(* CoDeSys 2.3.9.28 project: md_roman_5.pro *)
(* Libraries: SysLibTime.lib 2.12.10 13:48:32, Building_common.lib 2.12.10 13:48:40, mod_com.lib 2.12.10 13:48:32, DaylightSaving.lib 2.12.10 13:48:32, PowerMeasurement_01.lib 28.1.08 13:32:32, ModbusEthernet_04.lib 2.12.10 13:48:36, Util.lib 18.5.10 14:14:28, Standard.lib 2.12.10 13:48:34, SYSLIBCALLBACK.LIB 2.12.10 13:48:32, SysLibRtc.lib 2.12.10 13:48:32, SysLibFile.lib 2.12.10 13:48:34, Visu_Scheduler_03_e.lib 15.3.11 07:49:24, Scheduler_03.lib 9.3.11 15:45:22, DALI_02.lib 19.10.11 13:30:12, WagoLibDaylightSaving.lib 2.12.10 13:48:32, Ethernet.lib 2.12.10 13:48:32 *)

(* PLC configuration (modules and I/O channels)
TL01 AT %IX17.0 [BOOLOnX_I] Vypinac_sklad_sklad
TL02 AT %IX17.1 [BOOLOnX_I] Vypinac_sklad_prodejna
TL03 AT %IX17.2 [BOOLOnX_I] Vypinac_sklad_z_venku
TL04 AT %IX17.3 [BOOLOnX_I] Vypinac_sklad_vrata_predni
TL05 AT %IX17.4 [BOOLOnX_I] Vypinac_sklad_vrata_zadni
TL06 AT %IX17.5 [BOOLOnX_I] Vypinac_prodejna_kolotoc_sude
TL07 AT %IX17.6 [BOOLOnX_I] Vypinac_prodejna_kolotoc_liche
TL08 AT %IX17.7 [BOOLOnX_I] Vypinac_prodejna_vypinac
TL09 AT %IX17.8 [BOOLOnX_I] Prodejna_Dali
TL10 AT %IX17.9 [BOOLOnX_I] Prodejna_faugule_OUT13
TL11 AT %IX17.10 [BOOLOnX_I] Ch_3 Digital input
TL12 AT %IX17.11 [BOOLOnX_I] Ch_4 Digital input
TL13 AT %IX17.12 [BOOLOnX_I] Ch_5 Digital input
AT %IX17.13 [BOOLOnX_I] Ch_6 Digital input
AT %IX17.14 [BOOLOnX_I] Ch_7 Digital input
AT %IX17.15 [BOOLOnX_I] Ch_8 Digital input
AT %IX18.0 [BOOLOnX_I] Ch_1 Digital input
AT %IX18.1 [BOOLOnX_I] Ch_2 Digital input
AT %IX18.2 [BOOLOnX_I] Ch_3 Digital input
AT %IX18.3 [BOOLOnX_I] Ch_4 Digital input
AT %IX18.4 [BOOLOnX_I] Ch_5 Digital input
AT %IX18.5 [BOOLOnX_I] Ch_6 Digital input
AT %IX18.6 [BOOLOnX_I] Ch_7 Digital input
AT %IX18.7 [BOOLOnX_I] Ch_8 Digital input
KA01 AT %QX9.0 [BOOLOnX_Q] Nevim
KA02 AT %QX9.1 [BOOLOnX_Q] kolotoc2
KA03 AT %QX9.2 [BOOLOnX_Q] kolotoc3
KA04 AT %QX9.3 [BOOLOnX_Q] kolotoc4
KA05 AT %QX9.4 [BOOLOnX_Q] kolotoc5
KA06 AT %QX9.5 [BOOLOnX_Q] kolotoc6
KA07 AT %QX9.6 [BOOLOnX_Q] kolotoc7
KA08 AT %QX9.7 [BOOLOnX_Q] kolotoc8
0750-0530 8 DO 24 V DC 0.5A [Type_10_8_Channels] node 4, in %IB4 out %QB4 {INTTypePAAssignment = PLC; INTTypeModule = plugged}
  KA09 AT %QX9.8 [BOOLOnX_Q] kolotoc9
  KA10 AT %QX9.9 [BOOLOnX_Q] kolotoc10
  KA11 AT %QX9.10 [BOOLOnX_Q] kolotoc11
  KA12 AT %QX9.11 [BOOLOnX_Q] kolotoc12
  KA13 AT %QX9.12 [BOOLOnX_Q] svetlo_vchod_do_prodejny
  KA14 AT %QX9.13 [BOOLOnX_Q] reklama
  KA15 AT %QX9.14 [BOOLOnX_Q] svetlo_vrata_predni
  KA16 AT %QX9.15 [BOOLOnX_Q] svetlo_vrata_zadni
0750-0530 8 DO 24 V DC 0.5A [Type_10_8_Channels] node 5, in %IB5 out %QB5 {INTTypePAAssignment = PLC; INTTypeModule = plugged}
  KA17 AT %QX10.0 [BOOLOnX_Q] Ch_1 Digital output
  AT %QX10.1 [BOOLOnX_Q] Ch_2 Digital output
  AT %QX10.2 [BOOLOnX_Q] Ch_3 Digital output
  KA20 AT %QX10.3 [BOOLOnX_Q] Ch_4 Digital output
  AT %QX10.4 [BOOLOnX_Q] Ch_5 Digital output
  AT %QX10.5 [BOOLOnX_Q] Ch_6 Digital output
  AT %QX10.6 [BOOLOnX_Q] Ch_7 Digital output
  AT %QX10.7 [BOOLOnX_Q] Ch_8 Digital output
0750-0530 8 DO 24 V DC 0.5A [Type_10_8_Channels] node 6, in %IB6 out %QB6 {INTTypePAAssignment = PLC; INTTypeModule = plugged}
  AT %QX10.8 [BOOLOnX_Q] Ch_1 Digital output
  AT %QX10.9 [BOOLOnX_Q] Ch_2 Digital output
  AT %QX10.10 [BOOLOnX_Q] Ch_3 Digital output
  AT %QX10.11 [BOOLOnX_Q] Ch_4 Digital output
  AT %QX10.12 [BOOLOnX_Q] Ch_5 Digital output
  AT %QX10.13 [BOOLOnX_Q] Ch_6 Digital output
  AT %QX10.14 [BOOLOnX_Q] Ch_7 Digital output
  AT %QX10.15 [BOOLOnX_Q] Ch_8 Digital output
Analog_1 AT %IW0 [WORDOnW_I] Ch_1 Input word
AT %IW1 [WORDOnW_I] Ch_2 Input word
AT %IW2 [WORDOnW_I] Ch_3 Input word
AT %IW3 [WORDOnW_I] Ch_4 Input word
0750-0460/0000-0005 4 AI NI1000 (RTD) [Type_44_4_Channels] node 8, in %IB8 out %QB8 {INTTypePAAssignment = PLC; INTTypeModule = plugged}
  Teplota_1 AT %IW4 [INTOnW_I] Ch_1 signed Input value
  Teplota_2 AT %IW5 [INTOnW_I] Ch_2 signed Input value
  Teplota_3 AT %IW6 [INTOnW_I] Ch_3 signed Input value
  Teplota_4 AT %IW7 [INTOnW_I] Ch_4 signed Input value
0750-0641 DALI/DSI-Master [Type_36_1_Channels] node 9, in %IB9 out %QB9 {INTTypePAAssignment = PLC; INTTypeModule = plugged}
  AT %IX8.0 [BOOLOnX_I] Transmit accepted
  AT %IX8.1 [BOOLOnX_I] Receive request
  AT %IX8.2 [BOOLOnX_I] Init accepted
  AT %IX8.3 [BOOLOnX_I] Actor Error
  AT %IX8.4 [BOOLOnX_I] Frame Error
  AT %IX8.5 [BOOLOnX_I] Bus Error
  AT %IX8.6 [BOOLOnX_I] General Module Error
  AT %IB17 [BYTEOnB_I] DALI Response
  AT %IB18 [BYTEOnB_I] DALI Address
  AT %IB19 [BYTEOnB_I] Message 3
  AT %IB20 [BYTEOnB_I] Message 2
  AT %IB21 [BYTEOnB_I] Message 1
  AT %QX0.0 [BOOLOnX_Q] Transmit request
  AT %QX0.1 [BOOLOnX_Q] Receive accepted
  AT %QX0.2 [BOOLOnX_Q] Init request
  AT %QB1 [BYTEOnB_Q] DALI Command, DSI dimming value
  AT %QB2 [BYTEOnB_Q] DALI Address
  AT %QB3 [BYTEOnB_Q] Parameter 2
  AT %QB4 [BYTEOnB_Q] Parameter 1
  AT %QB5 [BYTEOnB_Q] Command extension
fazeVstup AT %IB22 [BYTEOnB_I] First Byte of 12
fazeVystup AT %QB6 [BYTEOnB_Q] First Byte of 12
Fieldbus variables [FB_VARS] node 1, in %IB0 out %QB0
*)

(* Task configuration *)
TASK hlavni (PRIORITY := 1, INTERVAL := T#20ms);
	PLC_PRG();
END_TASK
TASK Cas (PRIORITY := 15, INTERVAL := T#1000ms);
	LetniZimniCas();
	CasProg();
END_TASK

(* Global variable list: Global_Variables *)
VAR_GLOBAL
	start_bit: BOOL;
	Inicialiazace_DALI: BOOL;
	Inicializuj: BOOL;
	TL08s: BOOL;
	TL07s: BOOL;
	TL10s: BOOL;
	TL06s: BOOL;
	TL05s: BOOL;
	TL01s: BOOL;
	TL09s: BOOL;
	Cidlo: REAL;
	Uroven1: REAL := 3.5;
	Uroven2: REAL := 5;
	ZpozdeniCidla: BYTE := 10;
	Cidlo_zpozdene: REAL;

	CasDatumAktualni 	: DT;
	DenvTydnu			: BYTE;
	Leto 					: BOOL;
	sCasDatumAktualni 	: STRING[20];

	Uroven_reklama1: REAL := 1.5;

	VzdalenyVstup1: BOOL;
	VzdalenyVstup2: BOOL;
	VzdalenyVstup3: BOOL;
	VzdalenyVstup4: BOOL;
	VzdalenyVstup5: BOOL;
	VzdalenyVstup6: BOOL;
	VzdalenyVstup7: BOOL;
	VzdalenyVstup8: BOOL;
	VzdalenyVstup9: BOOL;
	VzdalenyVstup10: BOOL;
	VzdalenyVstup11: BOOL;
	VzdalenyVstup12: BOOL;
	VzdalenyVstup13: BOOL;
	VzdalenyVstup14: BOOL;
	VzdalenyVstup15: BOOL;
	VzdalenyVstup16: BOOL;

	VzdalenyVystup1: BOOL;
	VzdalenyVystup2: BOOL;
	VzdalenyVystup3: BOOL;
	VzdalenyVystup4: BOOL;
	VzdalenyVystup5: BOOL;
	VzdalenyVystup6: BOOL;
	VzdalenyVystup7: BOOL;
	VzdalenyVystup8: BOOL;
	VzdalenyVystup9: BOOL;
	VzdalenyVystup10: BOOL;
	VzdalenyVystup11: BOOL;
	VzdalenyVystup12: BOOL;
	VzdalenyVystup13: BOOL;
	VzdalenyVystup14: BOOL;
	VzdalenyVystup15: BOOL;
	VzdalenyVystup16: BOOL;

	VzdalenaTeplota1: WORD;
	VzdalenaTeplota2: WORD;
	VzdalenaTeplota3: WORD;
	VzdalenaTeplota4: WORD;

	IPSlaveProdejnaMaterial: STRING:= '192.168.111.202';

	INVnitrniSvetla1: BOOL;
	INVnitrniSvetla2: BOOL;
	INVnitrniSvetla3: BOOL;
	INVnitrniZasuvkyDenniProvoz: BOOL;
	INSvetloNadVchodem: BOOL;
	INVnitrniReklama: BOOL;
	INVenkovniReklama: BOOL;
	INTopeniOkap: BOOL;
	OUTVnitrniSvetla1: BOOL;		(*KA1*)
	OUTVnitrniSvetla2: BOOL;		(*KA2*)
	OUTVnitrniSvetla3: BOOL;		(*KA3*)
	OUTVnitrniReklama: BOOL;		(*KA4*)
	OUTVenkovniReklama1: BOOL;		(*KA5*)
	OUTVenkovniReklama2: BOOL;		(*KA6*)
	OUTVenkovniReklama3: BOOL;		(*KA7*)
	OUTSvetloNadVchodem: BOOL;		(*KA78*)
	OUTTopeniOkap1: BOOL;		(*KA9*)
	OUTTopeniOkap2: BOOL;		(*KA10*)
	OUTZasuvky1: BOOL;		(*KA11*)
	OUTZasuvky3: BOOL;		(*KA12*)
	OUTNouzoveOsvetleni: BOOL;		(*KA13*)
	OUTVnitrniZasuvkyDenniProvoz: BOOL;
	OUTVenkovniReklama: BOOL;
	OUTTopeniOkap: BOOL;

	INVenkovniTeplota: REAL;
END_VAR
VAR_GLOBAL RETAIN PERSISTENT
	typCasProg1: typScheduleWeekly;
	typCasProg2: typScheduleWeekly;

	typCasProg3: typScheduleWeekly;
	typCasProg4: typScheduleWeekly;

	typCasProg5: typScheduleWeekly;
	typCasProg6: typScheduleWeekly;
END_VAR

(* POU PLC_PRG, FBD *)
PROGRAM PLC_PRG
VAR
	cas_datum: CurTimeEx;
	System_cas: SysTime64;
	System_datum: SystemTimeDate;
	kolotoc1: kolotoc;
	kolotoc2: kolotoc;
	BLINK_nouzaky: BLINK;
	LibovolnyVystup: BOOL;
	komunikace: SlaveUDP_IO;

	Test: SlaveUDP_IO;
	sendStr: ARRAY [1..100] OF WORD;
	RecStr: ARRAY [1..100] OF WORD;

	Init: BOOL;
	NoError: BOOL;

	VzdaleneVstupy1: WORD_TO_BOOL_16b;
	VzdaleneVystupy1: BOOL_TO_WORD_16b;
END_VAR
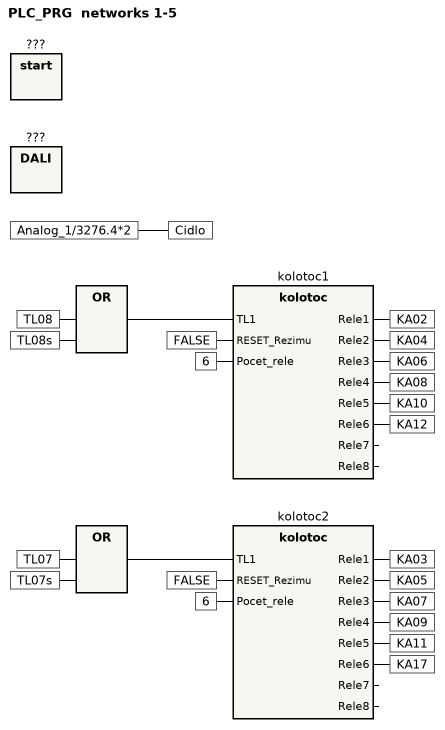
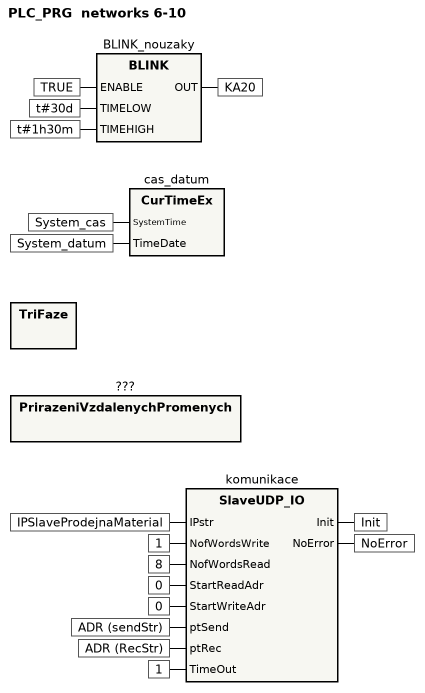
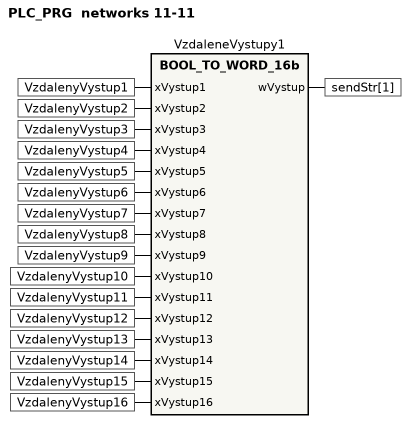
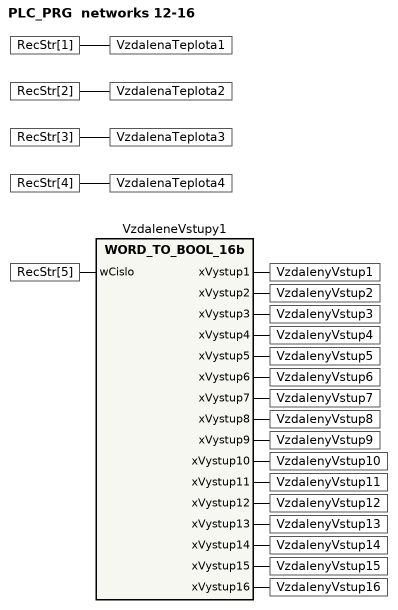
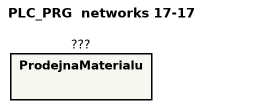
_FBD_ (* Function Block Diagram *)
NETWORK 1
	???:start()
NETWORK 2
	???:DALI()
NETWORK 3
	Analog_1/3276.4*2 => Cidlo
NETWORK 4
	kolotoc1:kolotoc(TL1: OR(TL08, TL08s), RESET_Rezimu: FALSE, Pocet_rele: 6, Rele2 => KA04, Rele3 => KA06, Rele4 => KA08, Rele5 => KA10, Rele6 => KA12) => KA02
NETWORK 5
	kolotoc2:kolotoc(TL1: OR(TL07, TL07s), RESET_Rezimu: FALSE, Pocet_rele: 6, Rele2 => KA05, Rele3 => KA07, Rele4 => KA09, Rele5 => KA11, Rele6 => KA17) => KA03
NETWORK 6
	BLINK_nouzaky:BLINK(ENABLE: TRUE, TIMELOW: t#30d, TIMEHIGH: t#1h30m) => KA20
NETWORK 7
	cas_datum:CurTimeEx(SystemTime: System_cas, TimeDate: System_datum)
NETWORK 8
	TriFaze()
NETWORK 9
	???:PrirazeniVzdalenychPromenych()
NETWORK 10
	komunikace:SlaveUDP_IO(IPstr: IPSlaveProdejnaMaterial, NofWordsWrite: 1, NofWordsRead: 8, StartReadAdr: 0, StartWriteAdr: 0, ptSend: ADR (sendStr), ptRec: ADR (RecStr), TimeOut: 1, NoError => NoError) => Init
NETWORK 11
	VzdaleneVystupy1:BOOL_TO_WORD_16b(xVystup1: VzdalenyVystup1, xVystup2: VzdalenyVystup2, xVystup3: VzdalenyVystup3, xVystup4: VzdalenyVystup4, xVystup5: VzdalenyVystup5, xVystup6: VzdalenyVystup6, xVystup7: VzdalenyVystup7, xVystup8: VzdalenyVystup8, xVystup9: VzdalenyVystup9, xVystup10: VzdalenyVystup10, xVystup11: VzdalenyVystup11, xVystup12: VzdalenyVystup12, xVystup13: VzdalenyVystup13, xVystup14: VzdalenyVystup14, xVystup15: VzdalenyVystup15, xVystup16: VzdalenyVystup16) => sendStr[1]
NETWORK 12
	RecStr[1] => VzdalenaTeplota1
NETWORK 13
	RecStr[2] => VzdalenaTeplota2
NETWORK 14
	RecStr[3] => VzdalenaTeplota3
NETWORK 15
	RecStr[4] => VzdalenaTeplota4
NETWORK 16
	VzdaleneVstupy1:WORD_TO_BOOL_16b(wCislo: RecStr[5], xVystup2 => VzdalenyVstup2, xVystup3 => VzdalenyVstup3, xVystup4 => VzdalenyVstup4, xVystup5 => VzdalenyVstup5, xVystup6 => VzdalenyVstup6, xVystup7 => VzdalenyVstup7, xVystup8 => VzdalenyVstup8, xVystup9 => VzdalenyVstup9, xVystup10 => VzdalenyVstup10, xVystup11 => VzdalenyVstup11, xVystup12 => VzdalenyVstup12, xVystup13 => VzdalenyVstup13, xVystup14 => VzdalenyVstup14, xVystup15 => VzdalenyVstup15, xVystup16 => VzdalenyVstup16) => VzdalenyVstup1
NETWORK 17
	???:ProdejnaMaterialu()
_END_FBD_
(* the same logic as Structured Text *)
(* Network 1: see the listing above *)
(* Network 2: see the listing above *)
(* Network 3 *)
Cidlo := Analog_1/3276.4*2;
(* Network 4 *)
kolotoc1(TL1 := TL08 OR TL08s, RESET_Rezimu := FALSE, Pocet_rele := 6);
KA04 := kolotoc1.Rele2;
KA06 := kolotoc1.Rele3;
KA08 := kolotoc1.Rele4;
KA10 := kolotoc1.Rele5;
KA12 := kolotoc1.Rele6;
KA02 := kolotoc1.Rele1;
(* Network 5 *)
kolotoc2(TL1 := TL07 OR TL07s, RESET_Rezimu := FALSE, Pocet_rele := 6);
KA05 := kolotoc2.Rele2;
KA07 := kolotoc2.Rele3;
KA09 := kolotoc2.Rele4;
KA11 := kolotoc2.Rele5;
KA17 := kolotoc2.Rele6;
KA03 := kolotoc2.Rele1;
(* Network 6 *)
BLINK_nouzaky(ENABLE := TRUE, TIMELOW := t#30d, TIMEHIGH := t#1h30m);
KA20 := BLINK_nouzaky.OUT;
(* Network 7 *)
cas_datum(SystemTime := System_cas, TimeDate := System_datum);
(* Network 8 *)
TriFaze();
(* Network 9: see the listing above *)
(* Network 10 *)
komunikace(IPstr := IPSlaveProdejnaMaterial, NofWordsWrite := 1, NofWordsRead := 8, StartReadAdr := 0, StartWriteAdr := 0, ptSend := ADR (sendStr), ptRec := ADR (RecStr), TimeOut := 1);
NoError := komunikace.NoError;
Init := komunikace.Init;
(* Network 11 *)
VzdaleneVystupy1(xVystup1 := VzdalenyVystup1, xVystup2 := VzdalenyVystup2, xVystup3 := VzdalenyVystup3, xVystup4 := VzdalenyVystup4, xVystup5 := VzdalenyVystup5, xVystup6 := VzdalenyVystup6, xVystup7 := VzdalenyVystup7, xVystup8 := VzdalenyVystup8, xVystup9 := VzdalenyVystup9, xVystup10 := VzdalenyVystup10, xVystup11 := VzdalenyVystup11, xVystup12 := VzdalenyVystup12, xVystup13 := VzdalenyVystup13, xVystup14 := VzdalenyVystup14, xVystup15 := VzdalenyVystup15, xVystup16 := VzdalenyVystup16);
sendStr[1] := VzdaleneVystupy1.wVystup;
(* Network 12 *)
VzdalenaTeplota1 := RecStr[1];
(* Network 13 *)
VzdalenaTeplota2 := RecStr[2];
(* Network 14 *)
VzdalenaTeplota3 := RecStr[3];
(* Network 15 *)
VzdalenaTeplota4 := RecStr[4];
(* Network 16 *)
VzdaleneVstupy1(wCislo := RecStr[5]);
VzdalenyVstup2 := VzdaleneVstupy1.xVystup2;
VzdalenyVstup3 := VzdaleneVstupy1.xVystup3;
VzdalenyVstup4 := VzdaleneVstupy1.xVystup4;
VzdalenyVstup5 := VzdaleneVstupy1.xVystup5;
VzdalenyVstup6 := VzdaleneVstupy1.xVystup6;
VzdalenyVstup7 := VzdaleneVstupy1.xVystup7;
VzdalenyVstup8 := VzdaleneVstupy1.xVystup8;
VzdalenyVstup9 := VzdaleneVstupy1.xVystup9;
VzdalenyVstup10 := VzdaleneVstupy1.xVystup10;
VzdalenyVstup11 := VzdaleneVstupy1.xVystup11;
VzdalenyVstup12 := VzdaleneVstupy1.xVystup12;
VzdalenyVstup13 := VzdaleneVstupy1.xVystup13;
VzdalenyVstup14 := VzdaleneVstupy1.xVystup14;
VzdalenyVstup15 := VzdaleneVstupy1.xVystup15;
VzdalenyVstup16 := VzdaleneVstupy1.xVystup16;
VzdalenyVstup1 := VzdaleneVstupy1.xVystup1;
(* Network 17: see the listing above *)
END_PROGRAM

(* POU dali/kolotoc, FBD *)
FUNCTION_BLOCK kolotoc
VAR
	Data_platna: BOOL;
	Data_platna_reset: BOOL;
	T_Data_platna: TON;
	T_Data_platna_reset: TON;
	Stisk_kratky: BOOL := FALSE;
	Stisk_dlouhy: BOOL := FALSE;
	T_stisk_TLx: TON;
	F_trig_hr1: F_TRIG;
	R_trig_hr2: R_TRIG;
	TL1_Citac: CTU;
	SR_stisk_TLx: SR;
	ZAP_VYP: BOOL;




	TP_byl_kratky: TP;
	Q_byl_kratky: BOOL;
	blok_kratky: BOOL;
	TL1_hr1: BOOL;
	SET_stisk_TL1: BOOL;
	Q_stisk_TL1: BOOL;
	TL1_INT: INT;
END_VAR

VAR_OUTPUT
	Rele1: BOOL;
	Rele2: BOOL;
	Rele3: BOOL;
	Rele4: BOOL;
	Rele5: BOOL;
	Rele6: BOOL;
	Rele7: BOOL;
	Rele8: BOOL;
END_VAR
VAR_INPUT
	TL1: BOOL;
	RESET_Rezimu: BOOL;
	Pocet_rele: INT;
END_VAR
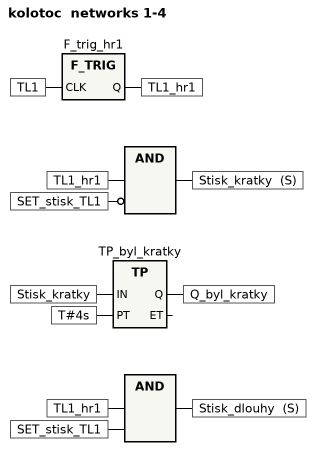
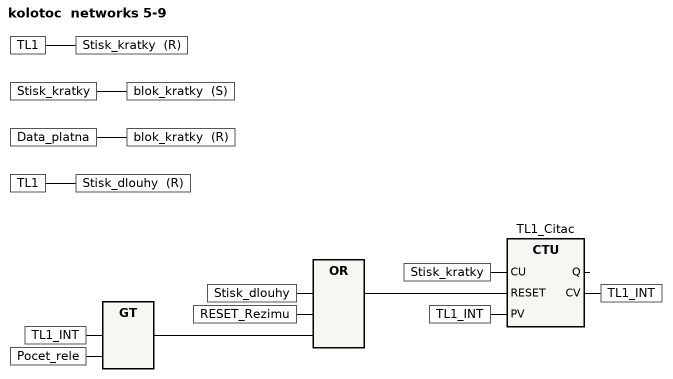
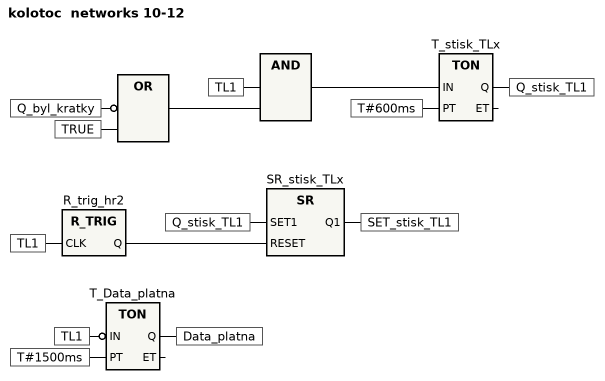
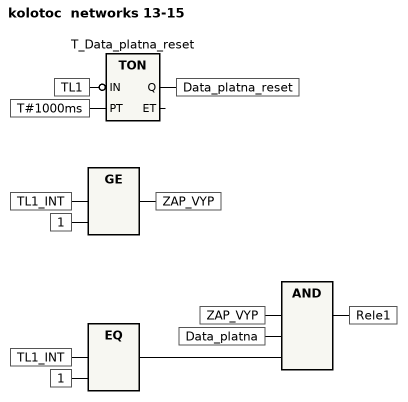
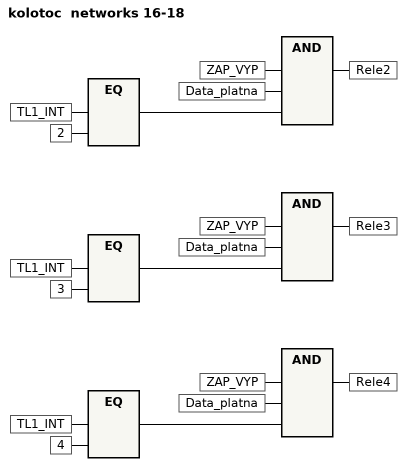
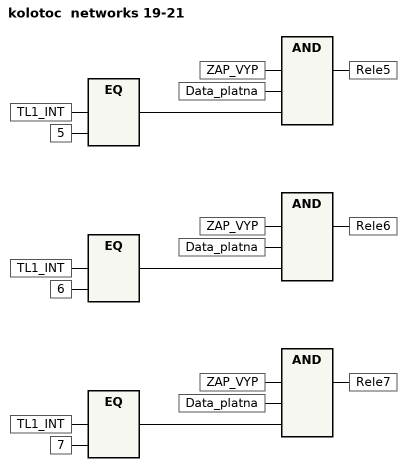
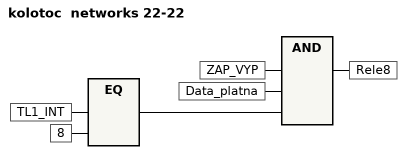
_FBD_ (* Function Block Diagram *)
NETWORK 1
	F_trig_hr1:F_TRIG(CLK: TL1) => TL1_hr1
NETWORK 2
	AND(TL1_hr1, NOT SET_stisk_TL1) => S Stisk_kratky
NETWORK 3
	TP_byl_kratky:TP(IN: Stisk_kratky, PT: T#4s) => Q_byl_kratky
NETWORK 4
	AND(TL1_hr1, SET_stisk_TL1) => S Stisk_dlouhy
NETWORK 5
	TL1 => R Stisk_kratky
NETWORK 6
	Stisk_kratky => S blok_kratky
NETWORK 7
	Data_platna => R blok_kratky
NETWORK 8
	TL1 => R Stisk_dlouhy
NETWORK 9
	TL1_Citac:CTU(CU: Stisk_kratky, RESET: OR(Stisk_dlouhy, RESET_Rezimu, GT(TL1_INT, Pocet_rele)), PV: TL1_INT, CV => TL1_INT)
NETWORK 10 (* delka stisku TLx *)
	T_stisk_TLx:TON(IN: AND(TL1, OR(NOT Q_byl_kratky, TRUE)), PT: T#600ms) => Q_stisk_TL1
NETWORK 11
	SR_stisk_TLx:SR(SET1: Q_stisk_TL1, RESET: R_trig_hr2:R_TRIG(CLK: TL1)) => SET_stisk_TL1
NETWORK 12 (* Data platna *)
	T_Data_platna:TON(IN: NOT TL1, PT: T#1500ms) => Data_platna
NETWORK 13 (* Data platna *)
	T_Data_platna_reset:TON(IN: NOT TL1, PT: T#1000ms) => Data_platna_reset
NETWORK 14
	GE(TL1_INT, 1) => ZAP_VYP
NETWORK 15
	AND(ZAP_VYP, Data_platna, EQ(TL1_INT, 1)) => Rele1
NETWORK 16
	AND(ZAP_VYP, Data_platna, EQ(TL1_INT, 2)) => Rele2
NETWORK 17
	AND(ZAP_VYP, Data_platna, EQ(TL1_INT, 3)) => Rele3
NETWORK 18
	AND(ZAP_VYP, Data_platna, EQ(TL1_INT, 4)) => Rele4
NETWORK 19
	AND(ZAP_VYP, Data_platna, EQ(TL1_INT, 5)) => Rele5
NETWORK 20
	AND(ZAP_VYP, Data_platna, EQ(TL1_INT, 6)) => Rele6
NETWORK 21
	AND(ZAP_VYP, Data_platna, EQ(TL1_INT, 7)) => Rele7
NETWORK 22
	AND(ZAP_VYP, Data_platna, EQ(TL1_INT, 8)) => Rele8
_END_FBD_
(* the same logic as Structured Text *)
(* Network 1 *)
F_trig_hr1(CLK := TL1);
TL1_hr1 := F_trig_hr1.Q;
(* Network 2 *)
IF TL1_hr1 AND NOT SET_stisk_TL1 THEN Stisk_kratky := TRUE; END_IF;
(* Network 3 *)
TP_byl_kratky(IN := Stisk_kratky, PT := T#4s);
Q_byl_kratky := TP_byl_kratky.Q;
(* Network 4 *)
IF TL1_hr1 AND SET_stisk_TL1 THEN Stisk_dlouhy := TRUE; END_IF;
(* Network 5 *)
IF TL1 THEN Stisk_kratky := FALSE; END_IF;
(* Network 6 *)
IF Stisk_kratky THEN blok_kratky := TRUE; END_IF;
(* Network 7 *)
IF Data_platna THEN blok_kratky := FALSE; END_IF;
(* Network 8 *)
IF TL1 THEN Stisk_dlouhy := FALSE; END_IF;
(* Network 9 *)
TL1_Citac(CU := Stisk_kratky, RESET := Stisk_dlouhy OR RESET_Rezimu OR (TL1_INT > Pocet_rele), PV := TL1_INT);
TL1_INT := TL1_Citac.CV;
(* Network 10: see the listing above *)
(* Network 11 *)
R_trig_hr2(CLK := TL1);
SR_stisk_TLx(SET1 := Q_stisk_TL1, RESET := R_trig_hr2.Q);
SET_stisk_TL1 := SR_stisk_TLx.Q1;
(* Network 12 *)
T_Data_platna(IN := NOT TL1, PT := T#1500ms);
Data_platna := T_Data_platna.Q;
(* Network 13 *)
T_Data_platna_reset(IN := NOT TL1, PT := T#1000ms);
Data_platna_reset := T_Data_platna_reset.Q;
(* Network 14 *)
ZAP_VYP := TL1_INT >= 1;
(* Network 15 *)
Rele1 := ZAP_VYP AND Data_platna AND (TL1_INT = 1);
(* Network 16 *)
Rele2 := ZAP_VYP AND Data_platna AND (TL1_INT = 2);
(* Network 17 *)
Rele3 := ZAP_VYP AND Data_platna AND (TL1_INT = 3);
(* Network 18 *)
Rele4 := ZAP_VYP AND Data_platna AND (TL1_INT = 4);
(* Network 19 *)
Rele5 := ZAP_VYP AND Data_platna AND (TL1_INT = 5);
(* Network 20 *)
Rele6 := ZAP_VYP AND Data_platna AND (TL1_INT = 6);
(* Network 21 *)
Rele7 := ZAP_VYP AND Data_platna AND (TL1_INT = 7);
(* Network 22 *)
Rele8 := ZAP_VYP AND Data_platna AND (TL1_INT = 8);
END_FUNCTION_BLOCK

(* POU SlaveUDP_IO, ST *)
FUNCTION_BLOCK SlaveUDP_IO
VAR_INPUT
	IPstr:STRING;					(*IP adresa slavu - 750-352,speedwaz etc.*)
	NofWordsWrite:WORD;		(*Pocet wordu, ktere maji byt zapsany*)
	NofWordsRead:WORD;		(*Pocet wordu, tkere maji byt cteny*)
	StartReadAdr:WORD;			(*adresa odkud se bude cist*)
	StartWriteAdr:WORD;			(*odresa kam se bude zapisovat*)
	ptSend:POINTER TO WORD;	(*pointer na pole ktere se bude zapisovat*)
	ptRec:POINTER TO WORD;	(*pointer na pole ktere se bude cist*)
	TimeOut:WORD:=500;		(*cas v milisekundach, pokud neni zadna komunikace, tak potomto case se vystupy nastavi do nuly*)
END_VAR
VAR_OUTPUT
	Init:BOOL;					(*cas do watchdogu byl zapsan a watchdog je spusten -> je mozne komunikovat*)
	NoError:BOOL;			(*zadna chyba pri komunikaci*)
END_VAR
VAR
	state:INT:=0;
	master882: ETHERNET_MODBUSMASTER_UDP;
	start882:BOOL:=FALSE;
	res882:BOOL:=FALSE;
	err882:WORD;
	ready882:BOOL;
	resp882:BYTE;
	ftrig882: F_TRIG;
	tmp_val:WORD;

	ptWrite:POINTER TO BYTE;
	NofWrite:INT;
	WriteAdr:WORD;
END_VAR
IF start882=FALSE THEN
	start882:=TRUE;
	CASE state OF
		0:
			(*zastaveni casovace*)
			tmp_val:=0;
			WriteAdr:=16#100A;
			ptWrite:=ADR(tmp_val);
			NofWrite:=1;
		1:
			(*nastaveni casu, cas je mozne nastavit jen tehdy, kdyz je casovac zastaven*)
			TimeOut:=TimeOut/100;
			tmp_val:=TimeOut;
			NofWordsWrite:=1;
			WriteAdr:=16#1000;
			ptWrite:=ADR(tmp_val);
			NofWrite:=1;
		2:
			(*spusteni watchdogu*)
			tmp_val:=1;
			WriteAdr:=16#100A;
			ptWrite:=ADR(tmp_val);
			NofWrite:=1;
		3:
			(*bezna komunikace*)
			ptWrite:=ptSend;
			NofWrite:=NofWordsWrite;
			WriteAdr:=StartWriteAdr;
	END_CASE;
END_IF;

NofWordsRead;
NofWrite;
IF NofWrite=0 THEN
(*cteni 352 kdyz neni treba nic zapsat*)
master882(strIP_ADDRESS := IPstr,	wPORT := 502,bUNIT_ID := 0,bFUNCTION_CODE := 3,wREAD_ADDRESS := StartReadAdr,wREAD_QUANTITY :=NofWordsRead,
	ptREAD_DATA :=ptRec,wWRITE_ADDRESS := WriteAdr,wWRITE_QUANTITY := NofWrite,ptSEND_DATA :=ptWrite ,xSTART := start882,xRESET := res882,
	tTIME_OUT := t#1s);
ELSE
(*blok pro cteni i zapis v jednom cyklu*)
master882(strIP_ADDRESS := IPstr,	wPORT := 502,bUNIT_ID := 0,bFUNCTION_CODE := 23,wREAD_ADDRESS := StartReadAdr,wREAD_QUANTITY :=NofWordsRead,
	ptREAD_DATA :=ptRec,wWRITE_ADDRESS := WriteAdr,wWRITE_QUANTITY := NofWrite,ptSEND_DATA :=ptWrite ,xSTART := start882,xRESET := res882,
	tTIME_OUT := t#1s);
END_IF;
	(* vystupni promenne *)
	err882:=master882.wERROR;
	ready882:= master882.xREADY;
	resp882:=master882.bRESPONSE_UNIT_ID;

IF master882.wERROR=0 THEN
	NoError:=TRUE;
ELSE
	NoError:=FALSE;
END_IF;
ftrig882(clk:=ready882);
(*prechody ve stavovem automau*)
IF ftrig882.Q   THEN
	 start882:=FALSE;
	IF master882.wERROR=0 THEN
		state:=state+1;	(*neni chyba komunikace, prejdi do dalsiho stavu*)
	ELSE
		IF state>0 AND state<3 THEN
			(*nastala nejaka chyba, vrat so inicializace casovace*)
			state:=0;
		END_IF;
	END_IF;
	IF state>=3 THEN
		state:=3;
		init:=TRUE;
	END_IF;
END_IF;
END_FUNCTION_BLOCK

(* POU Komunikace/WORD_TO_BOOL_16b, ST *)
FUNCTION_BLOCK WORD_TO_BOOL_16b
VAR_INPUT
	wCislo: WORD;

END_VAR
VAR_OUTPUT
	xVystup1: BOOL;
	xVystup2: BOOL;
	xVystup3: BOOL;
	xVystup4: BOOL;
	xVystup5: BOOL;
	xVystup6: BOOL;
	xVystup7: BOOL;
	xVystup8: BOOL;
	xVystup9: BOOL;
	xVystup10: BOOL;
	xVystup11: BOOL;
	xVystup12: BOOL;
	xVystup13: BOOL;
	xVystup14: BOOL;
	xVystup15: BOOL;
	xVystup16: BOOL;
END_VAR
VAR
END_VAR
IF (wCislo > 0)
	THEN
		(*15tý bit*)
		IF(wCislo/32768 > 0)
			THEN
				xVystup16 := TRUE;
				wCislo:= wCislo - 32768;
		ELSE
				xVystup16 := FALSE;
		END_IF

		(*14tý bit*)
		IF(wCislo/16384 > 0)
			THEN
				xVystup15 := TRUE;
				wCislo:= wCislo - 16384;
		ELSE
				xVystup15 := FALSE;
		END_IF

		(*13tý bit*)
		IF(wCislo/8192 > 0)
			THEN
				xVystup14 := TRUE;
				wCislo:= wCislo - 8192;
		ELSE
				xVystup14 := FALSE;
		END_IF

		(*12tý bit*)
		IF(wCislo/4096 > 0)
			THEN
				xVystup13 := TRUE;
				wCislo:= wCislo - 4096;
		ELSE
				xVystup13 := FALSE;
		END_IF

		(*11tý bit*)
		IF(wCislo/2048 > 0)
			THEN
				xVystup12 := TRUE;
				wCislo:= wCislo - 2048;
		ELSE
				xVystup12 := FALSE;
		END_IF

		(*10tý bit*)
		IF(wCislo/1024 > 0)
			THEN
				xVystup11 := TRUE;
				wCislo:= wCislo - 1024;
		ELSE
				xVystup11 := FALSE;
		END_IF

		(*9tý bit*)
		IF(wCislo/512 > 0)
			THEN
				xVystup10 := TRUE;
				wCislo:= wCislo - 512;
		ELSE
				xVystup10 := FALSE;
		END_IF

		(*8tý bit*)
		IF(wCislo/256 > 0)
			THEN
				xVystup9 := TRUE;
				wCislo:= wCislo - 256;
		ELSE
				xVystup9 := FALSE;
		END_IF

		(*7tý bit*)
		IF(wCislo/128 > 0)
			THEN
				xVystup8 := TRUE;
				wCislo:= wCislo - 128;
		ELSE
				xVystup8 := FALSE;
		END_IF

		(*6tý bit*)
		IF(wCislo/64 > 0)
			THEN
				xVystup7 := TRUE;
				wCislo:= wCislo - 64;
		ELSE
				xVystup7 := FALSE;
		END_IF

		(*5tý bit*)
		IF(wCislo/32 > 0)
			THEN
				xVystup6 := TRUE;
				wCislo:= wCislo - 32;
		ELSE
				xVystup6 := FALSE;
		END_IF

		(*4tý bit*)
		IF(wCislo/16 > 0)
			THEN
				xVystup5 := TRUE;
				wCislo:= wCislo - 16;
		ELSE
				xVystup5 := FALSE;
		END_IF

		(*3tí bit*)
		IF(wCislo/8 > 0)
			THEN
				xVystup4 := TRUE;
				wCislo:= wCislo - 8;
		ELSE
				xVystup4 := FALSE;
		END_IF

		(*2hý bit*)
		IF(wCislo/4 > 0)
			THEN
				xVystup3 := TRUE;
				wCislo:= wCislo - 4;
		ELSE
				xVystup3 := FALSE;
		END_IF

		(*1ní bit*)
		IF(wCislo/2 > 0)
			THEN
				xVystup2 := TRUE;
				wCislo:= wCislo - 2;
		ELSE
				xVystup2 := FALSE;
		END_IF

		(*0tý bit*)
		IF(wCislo > 0)
			THEN
				xVystup1 := TRUE;
				wCislo:= wCislo - 1;
		ELSE
				xVystup1 := FALSE;
		END_IF
ELSE
		xVystup1:= FALSE;
		xVystup2:= FALSE;
		xVystup3:= FALSE;
		xVystup4:= FALSE;
		xVystup5:= FALSE;
		xVystup6:= FALSE;
		xVystup7:= FALSE;
		xVystup8:= FALSE;
		xVystup9:= FALSE;
		xVystup10:= FALSE;
		xVystup11:= FALSE;
		xVystup12:= FALSE;
		xVystup13:= FALSE;
		xVystup14:= FALSE;
		xVystup15:= FALSE;
		xVystup16:= FALSE;
END_IF
END_FUNCTION_BLOCK

(* POU Komunikace/BOOL_TO_WORD_16b, CFC *)
FUNCTION_BLOCK BOOL_TO_WORD_16b
VAR_INPUT
	xVystup1: BOOL;
	xVystup2: BOOL;
	xVystup3: BOOL;
	xVystup4: BOOL;
	xVystup5: BOOL;
	xVystup6: BOOL;
	xVystup7: BOOL;
	xVystup8: BOOL;
	xVystup9: BOOL;
	xVystup10: BOOL;
	xVystup11: BOOL;
	xVystup12: BOOL;
	xVystup13: BOOL;
	xVystup14: BOOL;
	xVystup15: BOOL;
	xVystup16: BOOL;
END_VAR
VAR
END_VAR
VAR_OUTPUT
	wVystup: WORD;
END_VAR
VAR (* helpers for the ST form of the networks *)
	_t1 : WORD;
	_t8 : WORD;
	_t11 : WORD;
	_t14 : WORD;
	_t18 : WORD;
	_t21 : WORD;
	_t24 : WORD;
	_t27 : WORD;
	_t30 : WORD;
	_t33 : WORD;
	_t36 : WORD;
	_t39 : WORD;
	_t42 : WORD;
	_t45 : WORD;
	_t48 : WORD;
	_t6 : WORD;
END_VAR
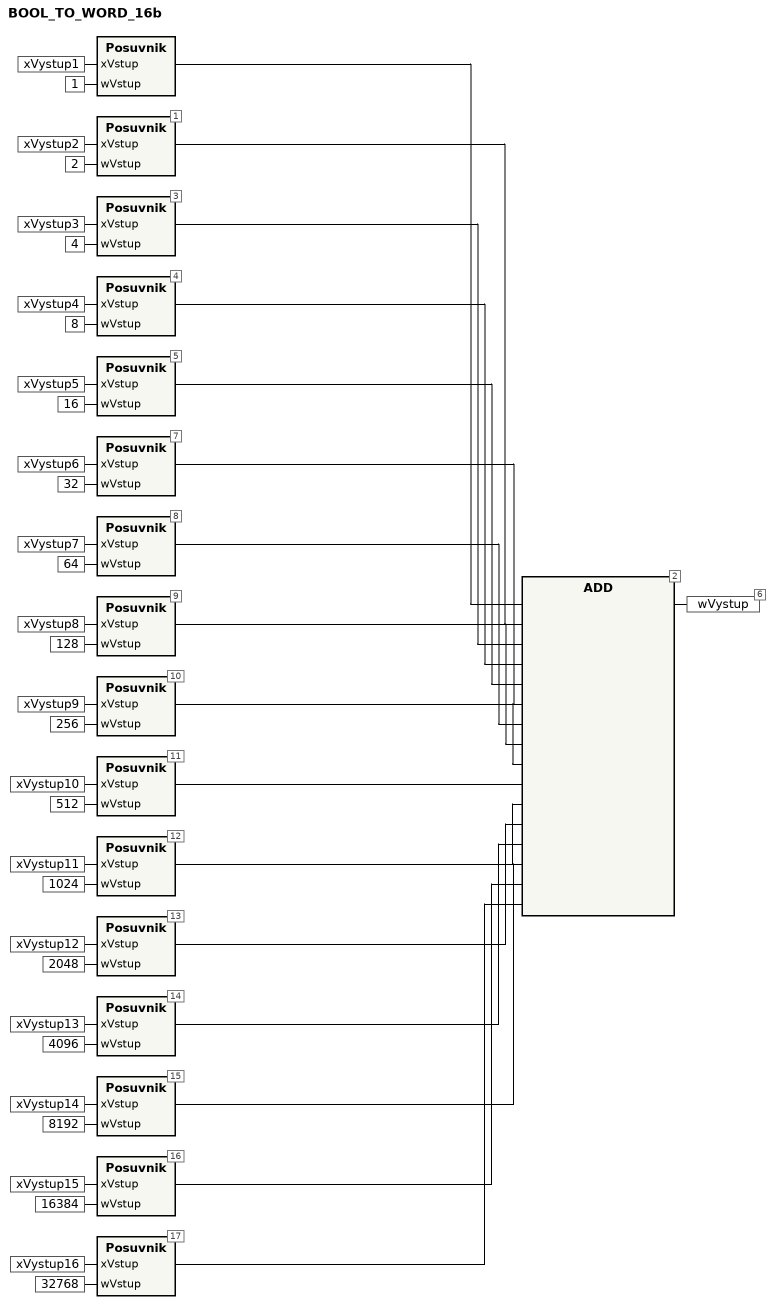
_CFC_ (* Continuous Function Chart, elements in execution order *)
#0 Posuvnik(xVstup: xVystup1, wVstup: 1)
#1 Posuvnik(xVstup: xVystup2, wVstup: 2)
#2 ADD(#0, #1, #3, #4, #5, #7, #8, #9, #10, #11, #12, #13, #14, #15, #16, #17)
#3 Posuvnik(xVstup: xVystup3, wVstup: 4)
#4 Posuvnik(xVstup: xVystup4, wVstup: 8)
#5 Posuvnik(xVstup: xVystup5, wVstup: 16)
#6 wVystup <= #2
#7 Posuvnik(xVstup: xVystup6, wVstup: 32)
#8 Posuvnik(xVstup: xVystup7, wVstup: 64)
#9 Posuvnik(xVstup: xVystup8, wVstup: 128)
#10 Posuvnik(xVstup: xVystup9, wVstup: 256)
#11 Posuvnik(xVstup: xVystup10, wVstup: 512)
#12 Posuvnik(xVstup: xVystup11, wVstup: 1024)
#13 Posuvnik(xVstup: xVystup12, wVstup: 2048)
#14 Posuvnik(xVstup: xVystup13, wVstup: 4096)
#15 Posuvnik(xVstup: xVystup14, wVstup: 8192)
#16 Posuvnik(xVstup: xVystup15, wVstup: 16384)
#17 Posuvnik(xVstup: xVystup16, wVstup: 32768)
_END_CFC_
(* the same logic as Structured Text *)
_t1 := Posuvnik(xVstup := xVystup1, wVstup := 1);
_t6 := _t1 + Posuvnik(xVstup := xVystup2, wVstup := 2) + _t8 + _t11 + _t14 + _t18 + _t21 + _t24 + _t27 + _t30 + _t33 + _t36 + _t39 + _t42 + _t45 + _t48;
_t8 := Posuvnik(xVstup := xVystup3, wVstup := 4);
_t11 := Posuvnik(xVstup := xVystup4, wVstup := 8);
_t14 := Posuvnik(xVstup := xVystup5, wVstup := 16);
wVystup := _t6;
_t18 := Posuvnik(xVstup := xVystup6, wVstup := 32);
_t21 := Posuvnik(xVstup := xVystup7, wVstup := 64);
_t24 := Posuvnik(xVstup := xVystup8, wVstup := 128);
_t27 := Posuvnik(xVstup := xVystup9, wVstup := 256);
_t30 := Posuvnik(xVstup := xVystup10, wVstup := 512);
_t33 := Posuvnik(xVstup := xVystup11, wVstup := 1024);
_t36 := Posuvnik(xVstup := xVystup12, wVstup := 2048);
_t39 := Posuvnik(xVstup := xVystup13, wVstup := 4096);
_t42 := Posuvnik(xVstup := xVystup14, wVstup := 8192);
_t45 := Posuvnik(xVstup := xVystup15, wVstup := 16384);
_t48 := Posuvnik(xVstup := xVystup16, wVstup := 32768);
END_FUNCTION_BLOCK

(* POU Komunikace/Posuvnik, ST *)
FUNCTION Posuvnik : WORD
VAR_INPUT
	xVstup: BOOL;
	wVstup: WORD;
END_VAR
VAR
END_VAR
IF (xVstup = TRUE)
THEN
Posuvnik := wVstup;
ELSE
Posuvnik := 0;
END_IF
END_FUNCTION

(* POU start, FBD *)
PROGRAM start
VAR
END_VAR
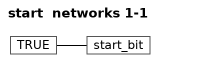
_FBD_ (* Function Block Diagram *)
NETWORK 1
	TRUE => start_bit
_END_FBD_
(* the same logic as Structured Text *)
(* Network 1 *)
start_bit := TRUE;
END_PROGRAM

(* POU dali/DALI, FBD *)
PROGRAM DALI
VAR
	trojklik_sklad: Trojklik;
	D_M: FbDALI_Joblist;

	Jobs: typDaliJoblisten;
	short_group: BOOL := FALSE;
	hodnota_po_zapnuti: BYTE := 50;
	hodnota_po_zapnuti_prodejna: BYTE := 100;
	povolit_vypnuti_pri_minimum: BOOL := FALSE;
	rychlost_zneny: BYTE := 7;
	co_je_kratky_a_dlouhy_stisk: TIME := t#600ms;
      OP_reset1: BOOL;
	OP_reset2: BOOL;
	OP_reset3: BOOL;
	OP_reset_OUT15: BOOL;
	OP_reset_OUT16: BOOL;

	Svetlo_adr1: FbDALI_LatchingRelay;
	Svetlo_adr2: FbDALI_LatchingRelay;
	Svetlo_adr3: FbDALI_LatchingRelay;
	Svetlo_adr4: FbDALI_DimmSingleButton;

	stav_adr1: BYTE;
	stav_adr2: BYTE;
	stav_adr3: BYTE;
	stav_adr4: BYTE;


	trojklik_prodejna: Trojklik;
	OP_reset4: BOOL;
	Trojklik_Fagule_OUT13: Trojklik;
	OP_reset5: BOOL;
	TP_ALL: TP;
	Q_All: BOOL;
	Dali_Status_03: FbDALI_StatusDimmValue;
	dali_status_Ready03: BOOL;
	dali_status_Feedback03: BYTE;
	dali_status_Status03: BOOL;
	dali_DimmValue_Ready03: BYTE;
	Reset_ini: TON;
	Dali_Status_09: FbDALI_StatusDimmValue;
	dali_status_Ready09: BOOL;
	dali_status_Feedback09: BYTE;
	dali_status_Status09: BOOL;
	dali_DimmValue_Ready09: BYTE;
	Dali_Status_19: FbDALI_StatusDimmValue;
	dali_status_Ready19: BOOL;
	dali_status_Feedback19: BYTE;
	dali_status_Status19: BOOL;
	dali_DimmValue_Ready19: BYTE;
	TON_ALL: TON;
	pom1: BOOL;
	go: BOOL;


	Fb_ShortLong1: Fb_ShortLong;
	CTU1: CTU;
	R_TRIG1: R_TRIG;
	TP1: TP;
	F_TRIG1: F_TRIG;
	STAV: WORD;
	CasNaKlik: TIME := t#1s500ms;
	F_TRIG2: F_TRIG;
	R_TRIG2: R_TRIG;
	Zhasni1: Zhasni;
	F_TRIG3: F_TRIG;
	Fb_LatchingRelay1: Fb_LatchingRelay;
	KratkyKlik: BOOL;
	Fb_ShortLong2: Fb_ShortLong;
	Fb_LatchingRelay2: Fb_LatchingRelay;
	Fb_ShortLong3: Fb_ShortLong;
	KratkyKlikA: BOOL;
	KratkyKlikB: BOOL;
	KratkyKlikC: BOOL;
	Svetlo_adr_255: FbDALI_LatchingRelay;
	stav_adr255: BYTE;
	TON_Cental_Off: TON;
	R_TRIG6: R_TRIG;
	ka15cas: TON;
	ka15pink: TP;
	TL06p: BOOL;
	ka16cas: TON;
	ka16pink: TP;
	TL05p: BOOL;
	ka13cas: TON;
	ka13pink: TP;
 	TL10p: BOOL;
	casvensvetel: TIME:= t#10m;
	Svetlo_adr5: FbDALI_LatchingRelay;
	stav_adr5: BYTE;
	Svetlo_adr6: FbDALI_LatchingRelay;
	stav_adr6: BYTE;
	Ovladani: Ovladani_7_8_9;
	aaa: BOOL;
	Svetlo_adr7: FbDALI_LatchingRelay;
	stav_adr7: BYTE;
	Svetlo_adr8: FbDALI_LatchingRelay;
	stav_adr8: BYTE;
	Svetlo_adr9: FbDALI_LatchingRelay;
	stav_adr9: BYTE;
END_VAR
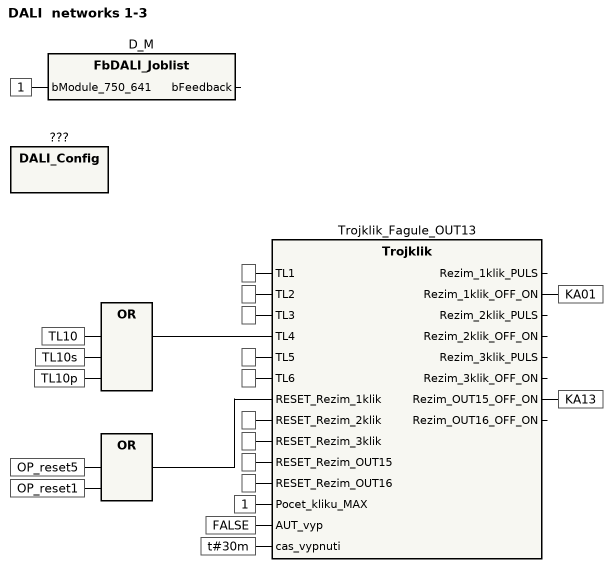
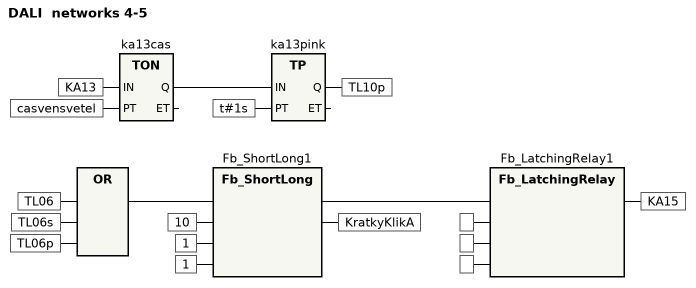
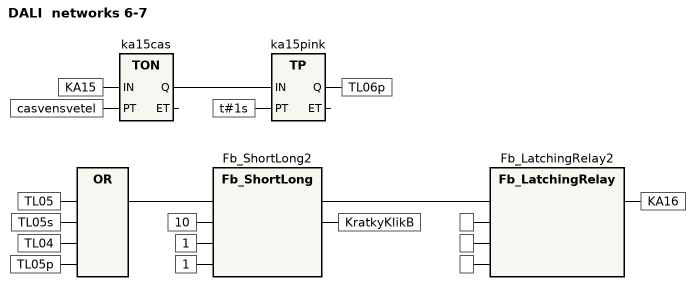
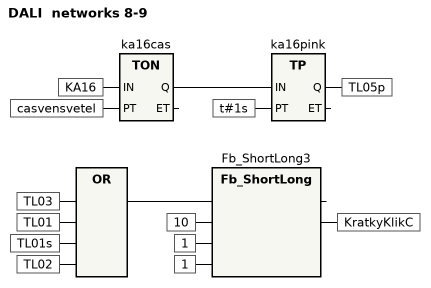
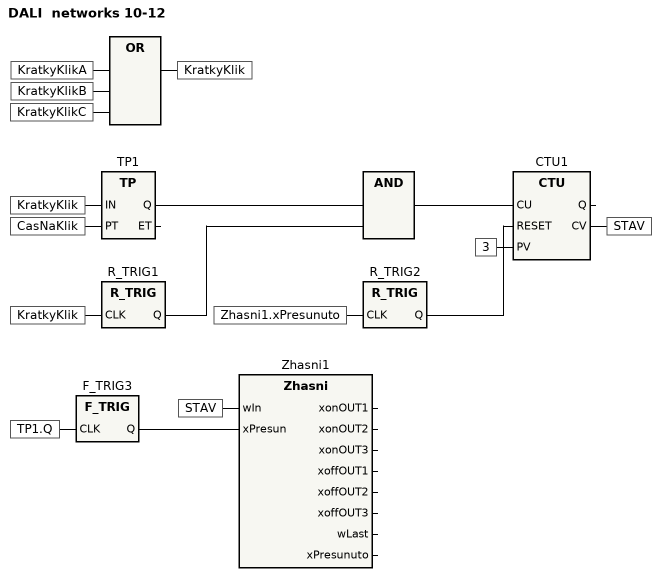
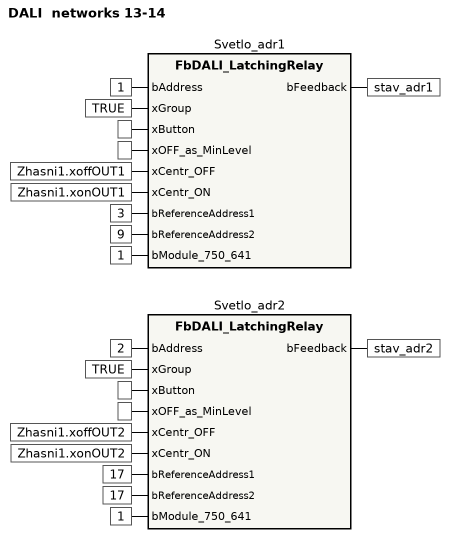
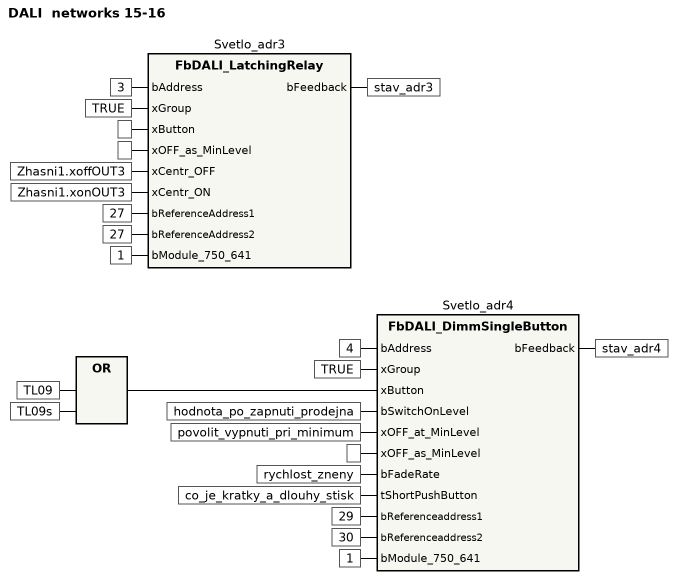
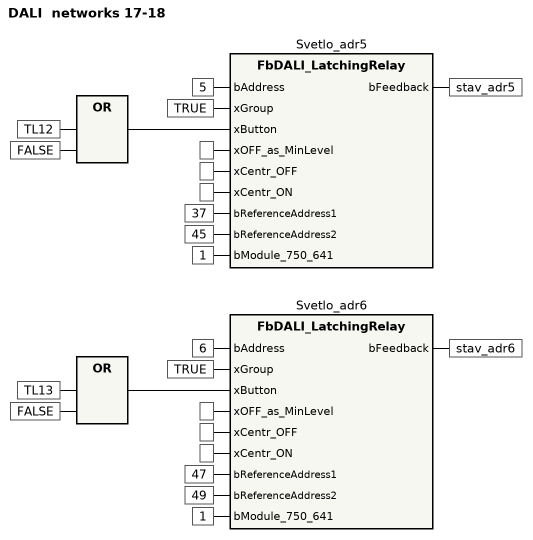
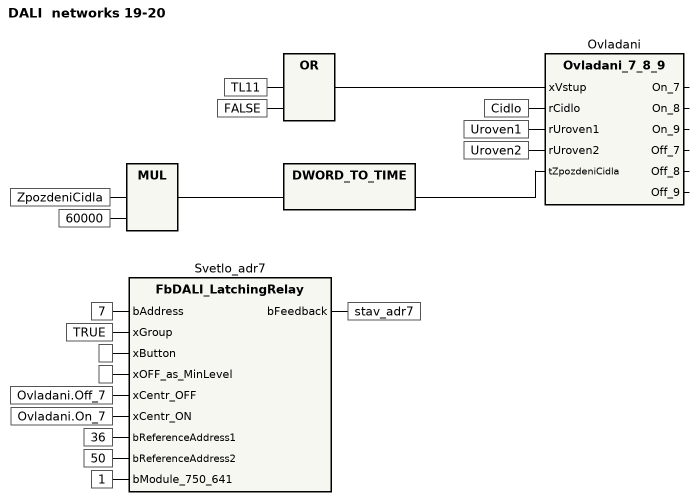
